// TIA Portal V19 export
DATA_BLOCK "ResetModules"   // DB4
// stored: InstanceOfName AFB_ResetModules, InstanceOfType FB
"AFB_ResetModules"
   // VAR
   //    c_vlv { S7_SetPoint := 'True'} : "C_VLV";
   //    c_cvlv { S7_SetPoint := 'True'} : "C_CVLV";
   //    c_mtr { S7_SetPoint := 'True'} : "C_MTR";
   //    c_mtrdir { S7_SetPoint := 'True'} : "C_MTRDIR";
   //    c_mtrlin { S7_SetPoint := 'True'} : "C_MTRLIN";
   // END_VAR
BEGIN
   c_vlv.enable := FALSE;
   c_vlv.index := 0;
   c_vlv.cmd := FALSE;
   c_vlv.upper := FALSE;
   c_vlv.lower := FALSE;
   c_vlv.blockMain := FALSE;
   c_vlv.blockUpper := FALSE;
   c_vlv.blockLower := FALSE;
   c_vlv.vfbMain := FALSE;
   c_vlv.hasJustAct := FALSE;
   c_vlv.vfbDeact := FALSE;
   c_vlv.hasjustDeact := FALSE;
   c_vlv.fault := FALSE;
   c_vlv.justHadFault := FALSE;
   c_vlv.justLostFault := FALSE;
   c_vlv.enabled := FALSE;
   c_vlv.auto := FALSE;
   c_vlv.status.isAct := FALSE;
   c_vlv.status.hasJustAct := FALSE;
   c_vlv.status.isDeact := FALSE;
   c_vlv.status.hasjustDeact := FALSE;
   c_vlv.status.inFault := FALSE;
   c_vlv.status.justHadFault := FALSE;
   c_vlv.status.justLostFault := FALSE;
   c_vlv.status.enabled := FALSE;
   c_vlv.status.auto := FALSE;
   c_vlv.status.old.position := FALSE;
   c_vlv.status.old.fault := FALSE;
   c_cvlv.enable := FALSE;
   c_cvlv.index := 0;
   c_cvlv.cmd := FALSE;
   c_cvlv.fup := FALSE;
   c_cvlv.status.running := FALSE;
   c_cvlv.status.justStarted := FALSE;
   c_cvlv.status.justStopped := FALSE;
   c_cvlv.status.reference := 0.0;
   c_cvlv.status.enabled := FALSE;
   c_cvlv.status.old.running := FALSE;
   c_mtr.enable := FALSE;
   c_mtr.index := 0;
   c_mtr.cmd := FALSE;
   c_mtr.block := FALSE;
   c_mtr.followUp := FALSE;
   c_mtr.spSource := FALSE;
   c_mtr.FUP := 0.0;
   c_mtr.SP := 0.0;
   c_mtr.PV := 0.0;
   c_mtr.PVunit := WSTRING#'';
   c_mtr.vfb := FALSE;
   c_mtr.fault := FALSE;
   c_mtr.justStarted := FALSE;
   c_mtr.justStopped := FALSE;
   c_mtr.justHadFault := FALSE;
   c_mtr.justLostFault := FALSE;
   c_mtr.enabled := FALSE;
   c_mtr.auto := FALSE;
   c_mtr.status.running := FALSE;
   c_mtr.status.inFault := FALSE;
   c_mtr.status.justStarted := FALSE;
   c_mtr.status.justStopped := FALSE;
   c_mtr.status.justHadFault := FALSE;
   c_mtr.status.justLostFault := FALSE;
   c_mtr.status.reference := 0.0;
   c_mtr.status.enabled := FALSE;
   c_mtr.status.auto := FALSE;
   c_mtr.status.old.running := FALSE;
   c_mtr.status.old.fault := FALSE;
   c_mtrdir.enable := FALSE;
   c_mtrdir.index := 0;
   c_mtrdir.cmd := FALSE;
   c_mtrdir.status.running := FALSE;
   c_mtrdir.status.inFault := FALSE;
   c_mtrdir.status.justStarted := FALSE;
   c_mtrdir.status.justStopped := FALSE;
   c_mtrdir.status.justHadFault := FALSE;
   c_mtrdir.status.justLostFault := FALSE;
   c_mtrdir.status.enabled := FALSE;
   c_mtrdir.status.old.running := FALSE;
   c_mtrdir.status.old.fault := FALSE;
   c_mtrlin.enable := FALSE;
   c_mtrlin.index := 0;
   c_mtrlin.cmd := FALSE;
   c_mtrlin.fup := FALSE;
   c_mtrlin.status.running := FALSE;
   c_mtrlin.status.inFault := FALSE;
   c_mtrlin.status.justStarted := FALSE;
   c_mtrlin.status.justStopped := FALSE;
   c_mtrlin.status.justHadFault := FALSE;
   c_mtrlin.status.justLostFault := FALSE;
   c_mtrlin.status.reference := 0.0;
   c_mtrlin.status.enabled := FALSE;
   c_mtrlin.status.old.running := FALSE;
   c_mtrlin.status.old.fault := FALSE;
END_DATA_BLOCK
